TYPE ST_OEE_In :
STRUCT
	Sec_PulseTrigger										: BOOL;
	Break_Active											: BOOL;
	EnableIn												: BOOL;	
	Select													: BOOL;
END_STRUCT
END_TYPE

(* stored: Version 1.1.0.1, ProductVersion 3.1.4024.2
   DUT ST_OEE_In: Id {60371e0d-96a2-4fae-a165-59aba8a034a2} *)
